ABB RobotStudio station: TicTacToe.rspag

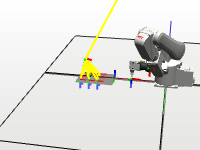
--- station ---
Station TicTacToe (saved by RobotStudio 6.7.7850.130)
Controller IRB_120_3kg_0.58m
  mechanical unit ROB_1: IRB120_3_58__01, 6 joints, base frame (0, 0, 0) mm
Layout (positions relative to the parent item):
  - IRB120_3_58__01 [mechanism, from Robots\IRB120_3_58_G_01.rslib] at (0, 0, 0) mm; joint values [0.9811, 0.9949, 1.2158, 1.2455, -1.78, 0.8008] (rad or m)
  - Pen [mechanism, from Training Objects\Pen.rslib] at (127.35, 70.3, 151.55) mm, rotated rx 95.78 ry 78.52 rz 83.89 deg
  - Pieza_4 [part] at (408.16, 128.97, 0) mm, rotated rx 0 ry 0 rz -90.26 deg
  - Sistema de coordenadas_1 [frame] at (408.43, 0, 0) mm
Attachment: Pen is attached to IRB120_3_58__01 / Link6
Targets, tools, work objects and paths stored in the station and not in the controller backup, written as RAPID:
! task T_ROB1
MODULE Module1
  CONST robtarget TRefContact_9_2:=[[128.032781484,-59.72,0.2],[0,0,1,0],[-1,-1,0,1],[9E+09,9E+09,9E+09,9E+09,9E+09,9E+09]];
ENDMODULE


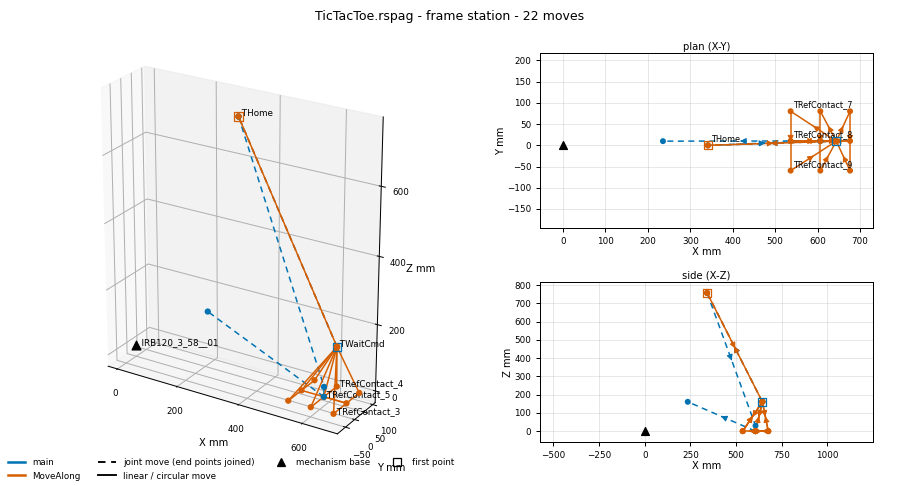
[picture p0: tool path of TicTacToe.rspag in frame station, 22 of 34 moves have a stored position in this frame; points joined in program order, loops and branches not executed]
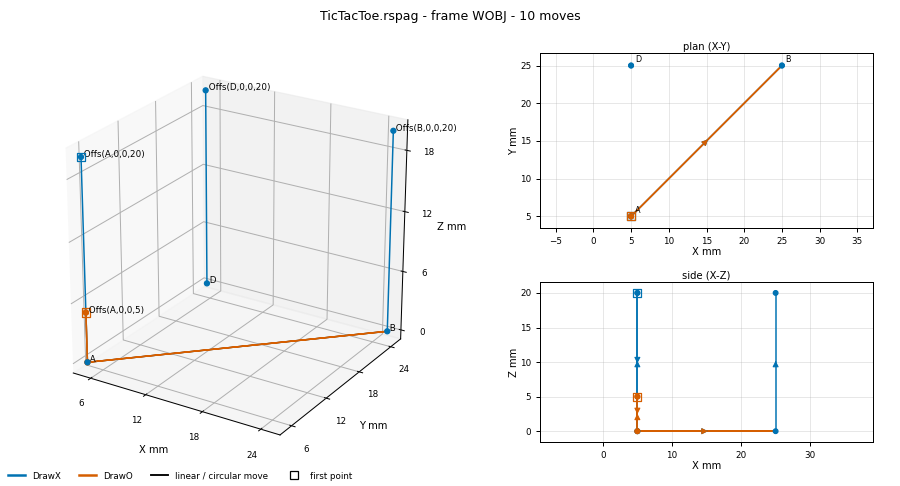
[picture p1: tool path of TicTacToe.rspag in frame WOBJ, 10 of 34 moves have a stored position in this frame; points joined in program order, loops and branches not executed]
--- Backups/IRB_120_3kg_0.58m/RAPID/TASK1/PROGMOD/CalibData.mod ---
MODULE CalibData
	TASK PERS wobjdata Workobject_1:=[FALSE,TRUE,"",[[408.434,0,0],[1,0,0,0]],[[0,0,0],[1,0,0,0]]];
    PERS tooldata Pen_TCP:=[TRUE,[[110,0,140],[0.707106781,0,0.707106781,0]],[1,[10.7435139,0,140],[1,0,0,0],0,0,0]];
ENDMODULE

--- Backups/IRB_120_3kg_0.58m/RAPID/TASK1/PROGMOD/MainModule.mod ---
MODULE MainModule
VAR socketdev server;
VAR socketdev client;
VAR string msg;
VAR rawbytes data;
 ! Array de 9 robtargets para una cuadrícula 3x3
  PERS wobjdata BASES{9};
  PERS wobjdata currentBase;
  ! Variables para cálculo
  PERS num GRID_SPACING := 50;  ! Separación de 50 mm
  CONST num OFFSET_X := 330.0;
  CONST num OFFSET_Y := 100.0;
    VAR string i;
    VAR string j;
    VAR string C;
    VAR num x;
    VAR num y;
    VAR num index;
    VAR bool ok;
  ! Rutina de inicialización de bases
  PROC InitGridBases()
    VAR num i;
    VAR num j;
    index:= 0;

    FOR i FROM 1 TO 3 DO  ! Filas
      FOR j FROM 1 TO 3 DO  ! Columnas
        index := (i-1) * 3 + j;  ! Índice en array

        ! Calcula coordenadas X e Y
        x := (j * GRID_SPACING);
        y := (i * GRID_SPACING);

        ! Asigna posición a la base
        BASES{index} :=[ FALSE, TRUE, "", [ [OFFSET_X, OFFSET_Y, 0], [1, 0, 0 ,0] ], [ [x, y, 0], [1, 0, 0 ,0] ] ];
      ENDFOR
    ENDFOR
  ENDPROC

PROC main()
    SocketCreate server;
    SocketBind server, "192.168.56.1", 5000;
    SocketListen server;
    SocketAccept server,client;

    InitGridBases;
    WHILE TRUE DO
        MoveJ TWaitCmd,v1000,z0,Pen_TCP \WObj:=Workobject_1;
        SocketReceive client, \str:=msg, \Time:=30;

        i := StrPart(msg,1,1);
        j := StrPart(msg,3,1);
        C := StrPart(msg,5,1);

        ok := StrToVal(i,x);
        ok := StrToVal(j,y);

        index := x * 3 + y + 1;
        currentBase :=[ FALSE, TRUE, "", [ [OFFSET_X, OFFSET_Y, 0], [1, 0, 0 ,0] ], [ [x*GRID_SPACING, y*GRID_SPACING, 0], [1, 0, 0 ,0] ] ];
        IF C = "X" THEN
            WaitUntil \inpos, TRUE;
            DrawX currentBase;
        ELSEIF C = "O" THEN
            MoveJ THome,v100,z0,Pen_TCP \WObj:=wobj0;
            MoveJ Offs(TRefContact_5,0,0,30),v1000,z1,Pen_TCP \WObj:=Workobject_1;
            MoveL TRefContact_5,v10,z0,Pen_TCP \WObj:=Workobject_1;
        ENDIF
        MoveJ TWaitCmd,v100,fine,Pen_TCP \WObj:=wobj0;

        SocketSend client,\Str:="DONE\0D\0A";
    ENDWHILE
    ERROR
        RETRY;
    UNDO
        SocketClose server;
        SocketClose client;
ENDPROC

PROC DrawX(PERS wobjdata WOBJ)

    VAR robtarget A := [ [5, 5, 0], [1, 0, 0, 0], [0, 0, 0, 0], [ 9E9, 9E9, 9E9, 9E9, 9E9, 9E9] ];
    VAR robtarget B := [ [25, 25, 0], [1, 0, 0, 0], [0, 0, 0, 0], [ 9E9, 9E9, 9E9, 9E9, 9E9, 9E9] ];
    VAR robtarget C := [ [25, 5, 0], [1, 0, 0, 0], [0, 0, 0, 0], [ 9E9, 9E9, 9E9, 9E9, 9E9, 9E9] ];
    VAR robtarget D := [ [5, 25, 0], [1, 0, 0, 0], [0, 0, 0, 0], [ 9E9, 9E9, 9E9, 9E9, 9E9, 9E9] ];


    MoveJ Offs(A,0,0,20), v100,z50,Pen_TCP \WObj:=WOBJ;
    WaitUntil \inpos, TRUE;
    MoveL A, v100,z50,Pen_TCP \WObj:=WOBJ;
    WaitUntil \inpos, TRUE;
    MoveL B, v100,z50,Pen_TCP \WObj:=WOBJ;
    WaitUntil \inpos, TRUE;
    MoveL Offs(B,0,0,20), v100,z50,Pen_TCP \WObj:=WOBJ;
    WaitUntil \inpos, TRUE;
    MoveJ Offs(C,0,0,20), v100,z50,Pen_TCP \WObj:=WOBJ;
    WaitUntil \inpos, TRUE;
    MoveL C, v100,z50,Pen_TCP \WObj:=WOBJ;
    WaitUntil \inpos, TRUE;
    MoveL D, v100,z50,Pen_TCP \WObj:=WOBJ;
    WaitUntil \inpos, TRUE;
    MoveL Offs(D,0,0,20), v100,z50,Pen_TCP \WObj:=WOBJ;
    WaitUntil \inpos, TRUE;
    WaitRob \ZeroSpeed;

ENDPROC

PROC DrawO(PERS wobjdata WOBJ)

    VAR robtarget A := [ [5, 5, 0], [1, 0, 0, 0], [1, 1, 0, 0], [ 9E9, 9E9, 9E9, 9E9, 9E9, 9E9] ];
    VAR robtarget B := [ [35, 35, 0], [1, 0, 0, 0], [1, 1, 0, 0], [ 9E9, 9E9, 9E9, 9E9, 9E9, 9E9] ];
    VAR robtarget D := [ [5, 25, 0], [1, 0, 0, 0], [1, 1, 0, 0], [ 9E9, 9E9, 9E9, 9E9, 9E9, 9E9] ];


    MoveJ Offs(A,0,0,5), v100,z50,Pen_TCP \WObj:=WOBJ;
     WaitUntil \inpos, TRUE;
    MoveL A, v100,z50,Pen_TCP \WObj:=WOBJ;
     WaitUntil \inpos, TRUE;
    MoveC B, A, v100,z50,Pen_TCP \WObj:=WOBJ;
     WaitUntil \inpos, TRUE;
    MoveL Offs(A,0,0,5), v100,z50,Pen_TCP \WObj:=WOBJ;
     WaitUntil \inpos, TRUE;
    WaitRob \ZeroSpeed;
     WaitUntil \inpos, TRUE;

ENDPROC
    PROC MoveAlong()
        MoveJ THome,v100,z0\Inpos:=stoptime0_5,Pen_TCP\WObj:=wobj0;
        MoveL TWaitCmd,v1000,z100,Pen_TCP\WObj:=Workobject_1;
        MoveL TRefContact_1,v1000,z100,Pen_TCP\WObj:=Workobject_1;
        MoveL TRefContact_3,v1000,z100,Pen_TCP\WObj:=Workobject_1;
        MoveL TWaitCmd,v1000,z100,Pen_TCP\WObj:=Workobject_1;
        MoveL TRefContact_4,v1000,z100,Pen_TCP\WObj:=Workobject_1;
        MoveL TRefContact_6,v1000,z100,Pen_TCP\WObj:=Workobject_1;
        MoveL TWaitCmd,v1000,z100,Pen_TCP\WObj:=Workobject_1;
        MoveL TRefContact_7,v1000,z100,Pen_TCP\WObj:=Workobject_1;
        MoveL TRefContact_9,v1000,z100,Pen_TCP\WObj:=Workobject_1;
        MoveL TWaitCmd,v1000,z100,Pen_TCP\WObj:=Workobject_1;
        MoveL TRefContact_5,v1000,z100,Pen_TCP\WObj:=Workobject_1;
        MoveL TRefContact_2,v1000,z100,Pen_TCP\WObj:=Workobject_1;
        MoveL TRefContact_5,v1000,z100,Pen_TCP\WObj:=Workobject_1;
        MoveL TRefContact_8,v1000,z100,Pen_TCP\WObj:=Workobject_1;
        MoveL TWaitCmd,v1000,z100,Pen_TCP\WObj:=Workobject_1;
        MoveJ THome,v100,z0\Inpos:=stoptime0_5,Pen_TCP\WObj:=wobj0;
    ENDPROC

ENDMODULE

--- Backups/IRB_120_3kg_0.58m/RAPID/TASK1/PROGMOD/Module1.mod ---
MODULE Module1
	CONST robtarget THome:=[[341.624381146,-0.149774337,756.856413922],[0.66065652,0.000489845,0.750478443,0.017743437],[0,0,0,1],[9E+09,9E+09,9E+09,9E+09,9E+09,9E+09]];
    CONST robtarget TRefContact_5:=[[198.032781484,10.28,0.2],[0,0,1,0],[0,0,-1,1],[9E+09,9E+09,9E+09,9E+09,9E+09,9E+09]];
    CONST robtarget TRefContact_1:=[[268.032781484,80.28,0.2],[0,0,1,0],[0,0,-1,1],[9E+09,9E+09,9E+09,9E+09,9E+09,9E+09]];
    CONST robtarget TRefContact_3:=[[268.032781484,-59.72,0.2],[0,0,1,0],[-1,-1,0,1],[9E+09,9E+09,9E+09,9E+09,9E+09,9E+09]];
    CONST robtarget TRefContact_9:=[[128.032781484,-59.72,0.2],[0,0,1,0],[-1,-1,0,1],[9E+09,9E+09,9E+09,9E+09,9E+09,9E+09]];
    CONST robtarget TRefContact_7:=[[128.032781484,80.28,0.2],[0,0,1,0],[0,0,-1,1],[9E+09,9E+09,9E+09,9E+09,9E+09,9E+09]];
    CONST robtarget TRefContact_2:=[[268.032781484,10.28,0.2],[0,0,1,0],[0,0,-1,1],[9E+09,9E+09,9E+09,9E+09,9E+09,9E+09]];
    CONST robtarget TRefContact_4:=[[198.032781484,80.28,0.2],[0,0,1,0],[0,0,-1,1],[9E+09,9E+09,9E+09,9E+09,9E+09,9E+09]];
    CONST robtarget TRefContact_6:=[[198.032781484,-59.72,0.2],[0,0,1,0],[-1,-1,0,1],[9E+09,9E+09,9E+09,9E+09,9E+09,9E+09]];
    CONST robtarget TRefContact_8:=[[128.032781484,10.28,0.2],[0,0,1,0],[0,0,-1,1],[9E+09,9E+09,9E+09,9E+09,9E+09,9E+09]];
    CONST robtarget TRefContact_5_2:=[[198.032781484,10.28,30.2],[0,0,1,0],[0,0,-1,1],[9E+09,9E+09,9E+09,9E+09,9E+09,9E+09]];
    CONST robtarget TWaitCmd:=[[235.608495677,9.73655562,160.901950418],[0.128841238,0.001247281,0.991653953,0.004562534],[0,0,-1,1],[9E+09,9E+09,9E+09,9E+09,9E+09,9E+09]];
ENDMODULE
